// TIA Portal V19 export
TYPE "LAF_typeSequence"
// Sequence data
// stored: Access Published
   STRUCT
      enableManualCtrl : Bool;   // Sequence can be controlled via hmiInteface
      enableManualModeChange : Bool;   // Mode of the sequence can changed via hmiInterface
      commands : "LAF_typeSequenceCommands";
      status { ExternalWritable := 'False'} : "LAF_typeSequenceStatus";
      previousSteps { ExternalWritable := 'False'} : Array[0..63] of "LAF_typeSequenceStep";   // History of the steps
   END_STRUCT;
END_TYPE
